FUNCTION_BLOCK AirSlider
VAR_INPUT CONSTANT
	bEnable : BOOL;
END_VAR
VAR_OUTPUT
	direction : AirMode;
	
	valveIn AT %Q* : BOOL;
	valveOut AT %Q* : BOOL;
	
	contact AT %I* : BOOL;
	
	home AT %I* : BOOL;
	innerLimit AT %I* : BOOL;
	
	ready : BOOL;
	busy : BOOL;
	error : BOOL;
	homeSet : BOOL;
END_VAR
VAR
	step : Homing;
END_VAR

IF NOT bEnable THEN
	valveIn := FALSE;
	valveOut := FALSE;
	RETURN;
END_IF

IF home OR innerLimit THEN
	direction := AirMode.HOLD;
END_IF

CASE direction OF
	AirMode.HOLD:
		valveIn := FALSE;
		valveOut := FALSE;
		
	AirMode.IN:
		valveIn := TRUE;
		valveOut := FALSE;
		
	AirMode.OUT:
		valveIn := FALSE;
		valveOut := TRUE;
		
END_CASE

METHOD homingSequence : BOOL
(*
this version of homing always traverses to the inner limit before returning to home,
eliminating the possibility of reaching the outer limit while homing
*)
CASE step OF
	Homing.IDLE:
		step := Homing.REDO;
		
	Homing.REDO: //technically HOME_IN, towards travel limit
		valveIn := TRUE;
		valveOut := FALSE;
		
		IF NOT innerLimit THEN
			valveIn := FALSE;
			valveOut := FALSE;
			step := Homing.HOME_OUT;
		END_IF
		
	Homing.HOME_OUT: //towards home
		valveIn := FALSE;
		valveOut := TRUE;
		
		IF NOT home THEN //if reached home
			valveIn := FALSE;
			valveOut := FALSE;
			step := Homing.DONE;
		END_IF
		
	Homing.DONE:
		valveIn := FALSE;
		valveOut := FALSE;
		homeSet := TRUE;
		
		homingSequence := TRUE;		
	
END_CASE
END_METHOD

METHOD slideIn : BOOL
VAR_INPUT
END_VAR
direction := AirMode.IN;

slideIn := TRUE;
END_METHOD

METHOD slideOut : BOOL
VAR_INPUT
END_VAR
direction := AirMode.OUT;

slideOut := TRUE;
END_METHOD

METHOD stop : BOOL
VAR_INPUT
END_VAR
valveIn := FALSE;
valveOut := FALSE;
direction := AirMode.HOLD;

stop := TRUE;
END_METHOD

END_FUNCTION_BLOCK

(* stored: Version 1.1.0.1, ProductVersion 3.1.4024.11
   POU AirSlider: Id {ef8d0471-4ac2-4d12-9e08-c4e8a3719cb6}, SpecialFunc None
   Method homingSequence: Id {c3ff30f8-ced2-4f8e-b758-e21ca109ec69}
   Method slideIn: Id {c905417d-ebb0-4426-b712-8b35f4512697}
   Method slideOut: Id {d6cfbb92-1846-4f17-b88f-dcdab10c19f1}
   Method stop: Id {c035c442-83bc-4f21-a06c-19730e7f9f48} *)
